   1:L PR[91] R[100]mm/sec CNT100;
   1:  PR[91,1] = PR[90,1] + 2.463;
   1:  PR[91,2] = PR[90,2] + 26.008;
   1:L PR[91] R[100]mm/sec CNT100 TB   .50sec,CALL END_PUD;
   1:  DO[117:Laser Start]=OFF;
   1:  PR[92] = PR[91];
   1:  PR[92,3] = PR[92,3] + 50;
   1:J PR[92] 10% FINE;
   1:  WAIT   5.00(sec);
   1:  DO[119:Gas]=OFF;
   1:  CALL HOME_ALL;
/POS
/END
